TYPE TAxisType :
	(	AT_Standard,
		AT_AX5000
	);
END_TYPE

(* stored: Version 1.1.0.1, ProductVersion 3.1.4022.12
   DUT TAxisType: Id {d644b4f6-5030-442a-b794-5e9aed13b4b5} *)
